(* IEC 61131-3 sources: ArfBotOS/Codesys-4/ArfBotOS.fbsdev/Application.iecapp^/FUN/tcp/FB_PythonServerHandler.fb.st^/P_Done.prop.st^, 1 file *)

(* ---- Get.meth.st ---- *)
VAR
END_VAR

P_Done := _Done;
